FUNCTION_BLOCK Test_F_NotEqual EXTENDS T_UnitTestBase
VAR
END_VAR

Assertion.AssertEquals_BOOL(
    Expected:= TRUE, 
    Actual:= F_NotEqual(1.000_005,1.000_003,0.000_001), 
    VariableName:= 'F_Equals');
    
Assertion.AssertEquals_BOOL(
    Expected:= FALSE, 
    Actual:= F_NotEqual(1.000_005,1.000_004,0.000_002), 
    VariableName:= 'F_Equals');
    
TestFinished();

END_FUNCTION_BLOCK

(* stored: Version 1.1.0.1, ProductVersion 3.1.4024.4
   POU Test_F_NotEqual: Id {337098c0-e2a6-447b-8374-90d85af5785b}, SpecialFunc None *)
